(**************************************************************************************
 * 	Application		:	BoxControl Framework
 *	Revision		:	$Revision: 404529 $
 *	Revision date	:	$Date: 2018-04-23 08:21:38 +0200 (Mo., 23 Apr 2018) $
 *	Last changed by	:	$Author: b7bolm $
 *	URL				:	$URL: http://almscdc.swisslog.com/repo/SWPD/Development/BoxControlFramework/20_Release/trunk/01_Software/BCF/BCF/JumpStart/20_Product/10_App/10_Base/10_Lib/00_GVLs/SDI_Table.TcGVL $
 *
 *	Purpose			:	SDO signals - separated due to debug reasons.
 *
 * ------------------------------------------------------------------------------------
 *	Copyright Swisslog [IP AG], Switzerland. All rights reserved.
 * 
 * ------------------------------------------------------------------------------------
 *	
 * 	Revision History: 
 *
 * 	VERSION			DATE			INITIALS			DESCRIPTION
 *	0.1				01.01.2001		swl					Example
 *
 **************************************************************************************)
VAR_GLOBAL CONSTANT
	NUMBER_OF_SDI_SIGNALS			: INT := 9999; // Number of SDI signals, max 9999 
END_VAR

VAR_GLOBAL
	SDISignalNumber					: ARRAY [0..NUMBER_OF_SDI_SIGNALS] OF ST_SDI_TABLE; // SDI table
END_VAR

(* stored: Version 1.1.0.1, ProductVersion 3.1.4022.12
   GVL SDI_Table: Id {22a85e74-7fdd-4fa7-8eaa-668e18c58215} *)
